PROGRAM MAIN
VAR
END_VAR

END_PROGRAM

(* stored: Version 1.1.0.1
   POU MAIN: Id {ed295dcb-e9ae-41f5-8c35-f2cb9f5cb69e} *)
